PROGRAM P_Demo_FB_HVACPriority_REAL_8
VAR
    fb : FB_HVACPriority_REAL_8;                            // 被演示 FB 实例
    eDataSecurityType_in : E_HVACDataSecurityType ;
    bEnable_in : BOOL := FALSE;
    eCtrlMode_in : E_HVACCtrlMode ;
    iManualValue_in : INT := 0;
    bDirection_in : BOOL := FALSE;
    rValueOut_out : REAL;
    bActive_out : BOOL;
    bEdgeNewEvent_out : BOOL;
    iValueNumber_out : INT;
END_VAR

// ============================================================================
// Tc2_HVAC.FB_HVACPriority_REAL_8 演示程序
// ============================================================================
// 场景：把本 FB 实例化到一个 PLC 程序里，每周期单次调用；按需要把 VAR_INPUT 与
//       VAR_IN_OUT 接到工程信号；VAR_OUTPUT 写入对应监视变量。
// 价值：使用本 FB 比手写状态机 / 控制算法节省大量代码；与 Tc2_HVAC 体系内其它 FB
//       直接对接，命名 / 持久化 / 模式仲裁等约定一致。具体语义见 FB_HVACPriority_REAL_8.md 主文档。
// 验证步骤：
//   1. 右键 PLC 项目下 POUs 文件夹 → Add → Existing Item → 选本 .TcPOU 文件
//   2. 引用 Tc2_HVAC（References → Add library）
//   3. 编译 → 登录 → 运行
//   4. 在线写各 *_in 输入信号触发 FB；在线 monitor *_out 引脚观察状态
// ============================================================================

fb(
    eDataSecurityType := eDataSecurityType_in,
    bEnable := bEnable_in,
    eCtrlMode := eCtrlMode_in,
    iManualValue := iManualValue_in,
    bDirection := bDirection_in,
    rValueOut => rValueOut_out,
    bActive => bActive_out,
    bEdgeNewEvent => bEdgeNewEvent_out,
    iValueNumber => iValueNumber_out
);

END_PROGRAM

(* stored: Version 1.1.0.1, ProductVersion 3.1.4024.5
   POU P_Demo_FB_HVACPriority_REAL_8: Id {823d29b4-4b3e-5106-b5f8-dd8fac8f6a96}, SpecialFunc None *)
